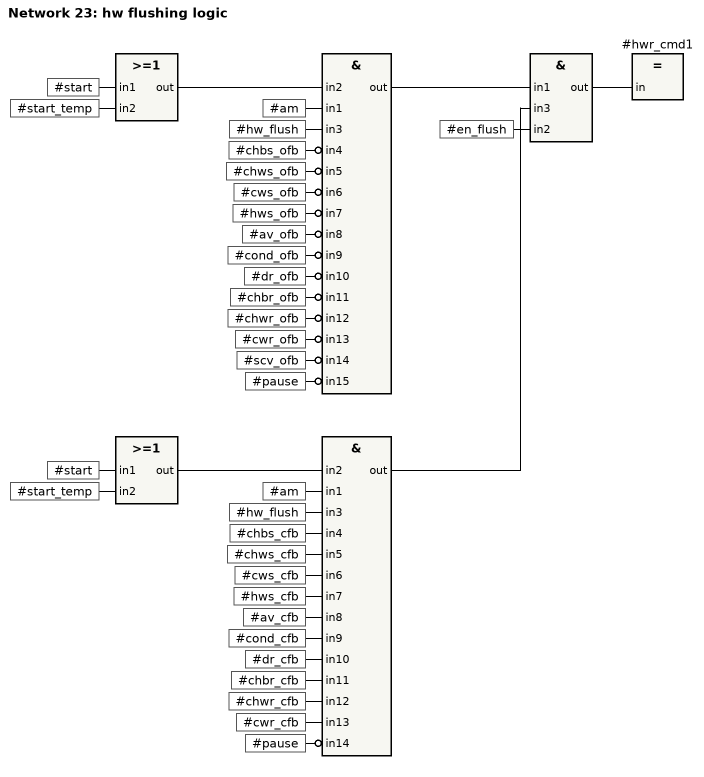
   #hwr_cmd1 := (#start OR #start_temp) AND #am AND #hw_flush AND NOT #chbs_ofb AND NOT #chws_ofb AND NOT #cws_ofb AND NOT #hws_ofb AND NOT #av_ofb AND NOT #cond_ofb AND NOT #dr_ofb AND NOT #chbr_ofb AND NOT #chwr_ofb AND NOT #cwr_ofb AND NOT #scv_ofb AND NOT #pause AND (#start OR #start_temp) AND #am AND #hw_flush AND #chbs_cfb AND #chws_cfb AND #cws_cfb AND #hws_cfb AND #av_cfb AND #cond_cfb AND #dr_cfb AND #chbr_cfb AND #chwr_cfb AND #cwr_cfb AND NOT #pause AND #en_flush;
END_REGION
END_FUNCTION_BLOCK
